FUNCTION_BLOCK FB_Bel_RGBW_Ablaufsteuerung
VAR_IN_OUT
	Zustand			: ST_Bel_Zustand;
	Stellwert		: ST_Bel_Stellwert;
END_VAR
VAR_INPUT
	Steuerung		: ST_Bel_Steuerung;
	Parameter		: ST_Bel_Parameter;
END_VAR
VAR_OUTPUT
END_VAR
VAR
	Timer: TON;
END_VAR

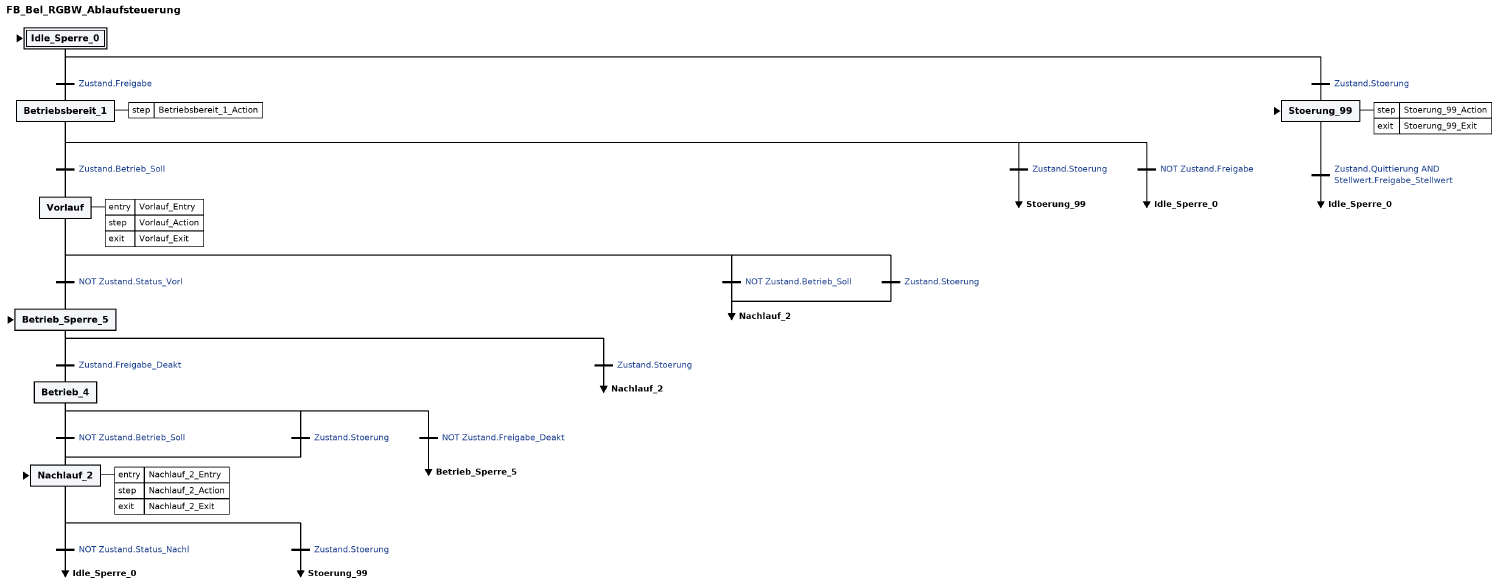
INITIAL_STEP Idle_Sperre_0:
END_STEP
TRANSITION FROM Idle_Sperre_0 TO Betriebsbereit_1
    := Zustand.Freigabe;
END_TRANSITION
TRANSITION FROM Idle_Sperre_0 TO Stoerung_99
    := Zustand.Stoerung;
END_TRANSITION
STEP Stoerung_99:
    Stoerung_99_Action(N);  // step action
    Stoerung_99_Exit(P0);  // exit action
END_STEP
TRANSITION FROM Stoerung_99 TO Idle_Sperre_0
    := Zustand.Quittierung AND Stellwert.Freigabe_Stellwert;
END_TRANSITION
STEP Betriebsbereit_1:
    Betriebsbereit_1_Action(N);  // step action
END_STEP
TRANSITION FROM Betriebsbereit_1 TO Vorlauf
    := Zustand.Betrieb_Soll;
END_TRANSITION
TRANSITION FROM Betriebsbereit_1 TO Stoerung_99
    := Zustand.Stoerung;
END_TRANSITION
TRANSITION FROM Betriebsbereit_1 TO Idle_Sperre_0
    := NOT Zustand.Freigabe;
END_TRANSITION
STEP Vorlauf:
    Vorlauf_Entry(P1);  // entry action
    Vorlauf_Action(N);  // step action
    Vorlauf_Exit(P0);  // exit action
END_STEP
TRANSITION FROM Vorlauf TO Betrieb_Sperre_5
    := NOT Zustand.Status_Vorl;
END_TRANSITION
TRANSITION FROM Vorlauf TO Nachlauf_2
    := NOT Zustand.Betrieb_Soll;
END_TRANSITION
TRANSITION FROM Vorlauf TO Nachlauf_2
    := Zustand.Stoerung;
END_TRANSITION
STEP Betrieb_Sperre_5:
END_STEP
TRANSITION FROM Betrieb_Sperre_5 TO Betrieb_4
    := Zustand.Freigabe_Deakt;
END_TRANSITION
TRANSITION FROM Betrieb_Sperre_5 TO Nachlauf_2
    := Zustand.Stoerung;
END_TRANSITION
STEP Betrieb_4:
END_STEP
TRANSITION FROM Betrieb_4 TO Nachlauf_2
    := NOT Zustand.Betrieb_Soll;
END_TRANSITION
TRANSITION FROM Betrieb_4 TO Nachlauf_2
    := Zustand.Stoerung;
END_TRANSITION
TRANSITION FROM Betrieb_4 TO Betrieb_Sperre_5
    := NOT Zustand.Freigabe_Deakt;
END_TRANSITION
STEP Nachlauf_2:
    Nachlauf_2_Entry(P1);  // entry action
    Nachlauf_2_Action(N);  // step action
    Nachlauf_2_Exit(P0);  // exit action
END_STEP
TRANSITION FROM Nachlauf_2 TO Idle_Sperre_0
    := NOT Zustand.Status_Nachl;
END_TRANSITION
TRANSITION FROM Nachlauf_2 TO Stoerung_99
    := Zustand.Stoerung;
END_TRANSITION

ACTION Betriebsbereit_1_Action:
Stellwert.Freigabe_Stellwert := TRUE;
END_ACTION

ACTION Nachlauf_2_Action:
(* Nachlauf Timer starten *)
Timer( 	IN := Zustand.Status_Nachl,
		PT := DINT_TO_TIME(Parameter.Zeit_Nachl)
);
Zustand.Status_Nachl	:= NOT(Timer.Q AND NOT Zustand.Betrieb);

(* Stellwert setzen *)
Stellwert.Betrieb := FALSE;
Stellwert.Freigabe_Stellwert := FALSE;

(* Zustand setzen *)
Zustand.Status := E_Bel_Zustand_Status_Nachl;
END_ACTION

ACTION Nachlauf_2_Entry:
Zustand.Status_Nachl := TRUE;
(* Reset Timer *)
Timer(IN := FALSE);
END_ACTION

ACTION Nachlauf_2_Exit:
Zustand.Status_Nachl := FALSE;
END_ACTION

ACTION Stoerung_99_Action:
(* Stellwert setzen *)
Stellwert.Betrieb := FALSE;

(* Zustand setzen *)
Zustand.Stoerung := TRUE;
Zustand.Status := E_Bel_Zustand_Status_Stoerung;
END_ACTION

ACTION Stoerung_99_Exit:
Zustand.Stoerung	:= FALSE;
END_ACTION

ACTION Vorlauf_Action:
(* Vorlaufzeit Timer starten *)
Timer( 	IN := Zustand.Status_Vorl,
		PT := DINT_TO_TIME(Parameter.Zeit_Vorl)
);
Zustand.Status_Vorl := NOT (Timer.Q AND Zustand.Betrieb);

(* Stellwert setzen *)
IF Stellwert.Freigabe_Stellwert = TRUE THEN
	Stellwert.Betrieb := TRUE;
END_IF

(* Zustand setzen *)
Zustand.Status := E_Bel_Zustand_Status_Vorl;
END_ACTION

ACTION Vorlauf_Entry:
Zustand.Status_Vorl := TRUE;
(* Reset Timer *)
Timer(IN := FALSE);
END_ACTION

ACTION Vorlauf_Exit:
Zustand.Status_Vorl := FALSE;
END_ACTION

END_FUNCTION_BLOCK

(* stored: Version 1.1.0.1, ProductVersion 3.1.4024.10
   POU FB_Bel_RGBW_Ablaufsteuerung: Id {e5e39f7a-704e-437d-b3ec-beb03bca0dc5}, SpecialFunc None
   Action Betriebsbereit_1_Action: Id {23b2ba9a-84cd-4fc8-90d5-8bb1559fdaab}
   Action Nachlauf_2_Action: Id {5683074a-fb8f-4862-b001-67877c3c99a4}
   Action Nachlauf_2_Entry: Id {d22a6478-b133-478f-a10c-a7aaaa81438b}
   Action Nachlauf_2_Exit: Id {c1be10b2-7f0a-4f36-8e45-5127a85c8fe5}
   Action Stoerung_99_Action: Id {b9383640-673b-4ff4-8e85-174bd3bde2c2}
   Action Stoerung_99_Exit: Id {7ccc040c-67c6-4e7a-81ea-389c4cd54de9}
   Action Vorlauf_Action: Id {fe74158a-c884-458e-9f5a-9e618aa248c1}
   Action Vorlauf_Entry: Id {f720664d-3f7d-420f-89a7-1d19bd83b8ba}
   Action Vorlauf_Exit: Id {9dbf4df4-fff4-447f-999e-0e74993b428a} *)
